TYPE ST_LogEntry :
STRUCT
    StationName  : STRING(40);
    StepNumber   : INT;
    CycleTimeMs  : LREAL;
    Timestamp    : DT;
END_STRUCT
END_TYPE

(* stored: Version 1.1.0.1
   DUT ST_LogEntry: Id {9d3c0cda-ecc7-49a6-ac4e-eec04a209cb5} *)
